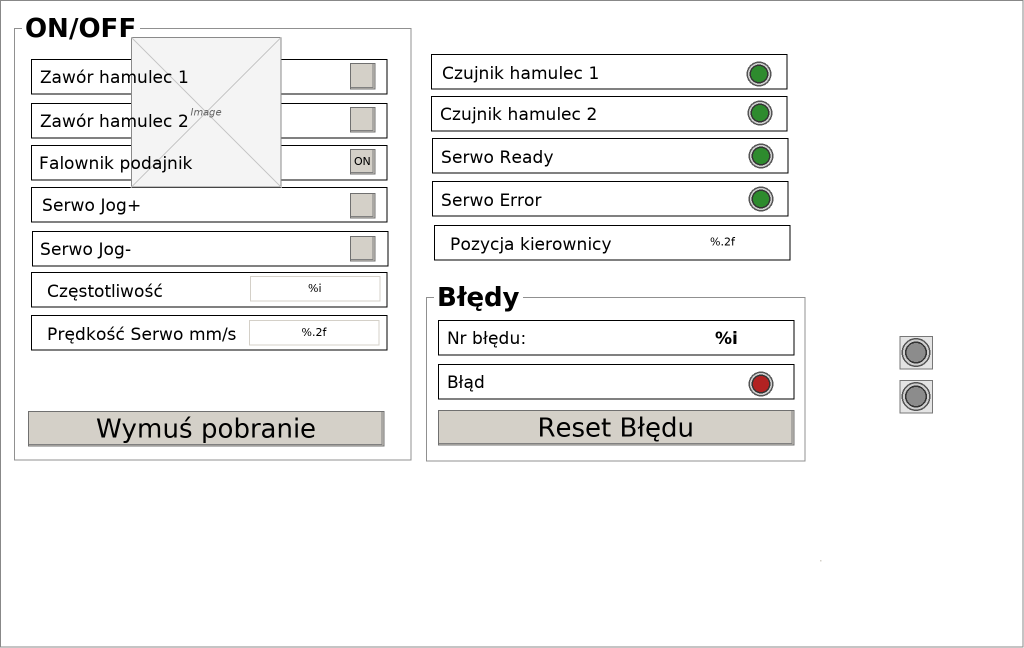
VISUALIZATION Kierwonica  // 1024x648
    Rectangle (31,59 356x35)
    Rectangle (31,103 356x35)
    Rectangle (31,145 356x35)
    Rectangle (31,272 356x35)
    Rectangle (32,231 356x35)
    Rectangle (31,187 356x35)
    GroupBox (14,20 397x440), "ON/OFF"
        Rectangle (17,295 356x35)
        Button (336,173 25x25)
            tap GVL_HMI.bHmiJogF
        Button (336,216 25x25)
            tap GVL_HMI.bHmiJogB
        Textfield (236,256 130x25), "%i", text variable: GVL_HMI.iFreqKierownicaMan
            OnMouseClick: write the text variable via Edit
        Button (336,129 25x25), "ON", colour toggle: GVL_GLOBAL.falownik_podajnik_kier_cewka
            tap GVL_HMI.przycisk_falownik_podajnik_kier
        Button (336,87 25x25), colour toggle: GVL_GLOBAL.zaw_ham2_kier_cewka
            tap GVL_HMI.przycisk_zaw_ham2_kier
        Button (336,43 25x26), colour toggle: GVL_GLOBAL.zaw_ham1_kier_cewka
            tap GVL_HMI.przycisk_zaw_ham1_kier
        Image (117,17 150x150)
        Button (14,391 356x35), "Wymuś pobranie"
            OnMouseDown: execute { GVL_HMI.Wymus_pobranie:=TRUE; }
    Rectangle (431,54 356x35)
    Label (437,57 230x30)
    Rectangle (431,96 356x35)
    Label (437,99 239x30), "Czujnik hamulec 2"
    Lamp1 (746,99 28x28), variable: GVL_IO_K.b4B6, style: Lamp-Lamp1-Green
    Lamp1 (745,60 28x28), variable: GVL_IO_K.b4B7, style: Lamp-Lamp1-Green
    Label (439,58 239x30), "Czujnik hamulec 1"
    Rectangle (432,138 356x35)
    Rectangle (432,181 356x35)
    Label (37,101 239x30)
    Label (37,106 209x30), "Zawór hamulec 2"
    Label (37,62 209x30), "Zawór hamulec 1"
    Label (36,148 209x30), "Falownik podajnik"
    Label (44,276 209x30), "Częstotliwość"
    Label (438,142 239x30), "Serwo Ready"
    Lamp1 (747,142 28x28), variable: PRG_Kierownica.S_K_Power.Status, style: Lamp-Lamp1-Green
    Label (438,185 239x30), "Serwo Error"
    Lamp1 (747,185 28x28), variable: PRG_Kierownica.S_K_Power.Error, style: Lamp-Lamp1-Green
    Rectangle (434,225 356x35)
    Label (447,229 209x30), "Pozycja kierownicy"
    Textfield (662,227 121x30), "%.2f", text variable: GVL_AXIS.stAxis2.NcToPlc.ActPos
    Label (39,190 209x30), "Serwo Jog+"
    Label (37,234 209x30), "Serwo Jog-"
    PushSwitch (897,380 38x33), behaviour: TOGGLE, style: Switch-PushSwitch-Gray
    PushSwitch (897,336 38x33), behaviour: TOGGLE, style: Switch-PushSwitch-Gray
    Textfield (249,320 130x25), "%.2f", text variable: gvl_hmi.J_Vel
        OnMouseClick: write the text variable via Edit
    Label (44,319 209x30), "Prędkość Serwo mm/s"
    Textfield (820,560 1x1)
    GroupBox (426,289 379x172), "Błędy"
        Rectangle (12,31 356x35)
        Label (18,34 209x30), "Nr błędu:"
        Rectangle (12,75 356x35)
        Label (18,78 209x30), "Błąd"
        Button (12,121 356x35), "Reset Błędu"
            tap GVL_HMI.ErrorResetKier
        Lamp1 (321,81 28x28), variable: GVL_GLOBAL.Error_pakowania, style: Lamp-Lamp1-Red
        Textfield (240,34 121x30), "%i", text variable: GVL_GLOBAL.Error_numb_kier
END_VISUALIZATION

(* stored: Version 1.1.0.1, ProductVersion 3.1.4022.12
   Visu Kierwonica: Id {9aaf6d74-8b6f-4b76-bc8e-8eae1d9546f8} *)
